(* Logix 5000 project; controller STAT 1756-L72 rev 20.12; software revision 20.04; part 29 of 34 *)
(* tags used below, declared in another part *)
   B3 : DINT[35];
   N20 : DINT[50];
   N7 : DINT[150];
   N9 : DINT[200];
   T4 : TIMER[100];
   comm : BOOL;
   L1_stat : DINT[20];
   L2_STAT : DINT[20];
   L3_STAT : DINT[20];
   lancystock1 : DINT;
   lancystock2 : DINT;
   N : INT[255];
   stat_L1 : DINT[20];
   STAT_L2 : DINT[20];
   STAT_L3 : DINT[20];
(* LANCY, continued *)

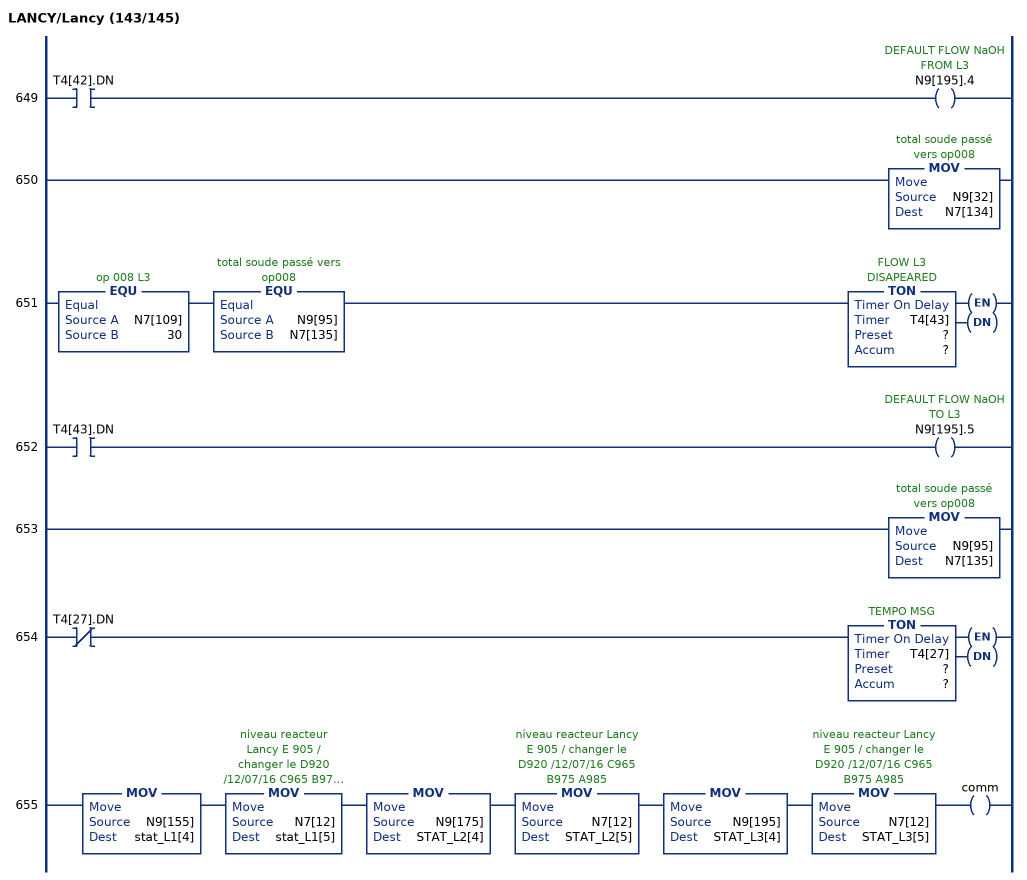
   649: XIC(T4[42].DN)OTE(N9[195].4);
   650: MOV(N9[32],N7[134]);
   651: EQU(N7[109],30)EQU(N9[95],N7[135])TON(T4[43],?,?);
   652: XIC(T4[43].DN)OTE(N9[195].5);
   653: MOV(N9[95],N7[135]);
   654: XIO(T4[27].DN)TON(T4[27],?,?);
   655: MOV(N9[155],stat_L1[4])MOV(N7[12],stat_L1[5])MOV(N9[175],STAT_L2[4])MOV(N7[12],STAT_L2[5])MOV(N9[195],STAT_L3[4])MOV(N7[12],STAT_L3[5])OTE(comm);
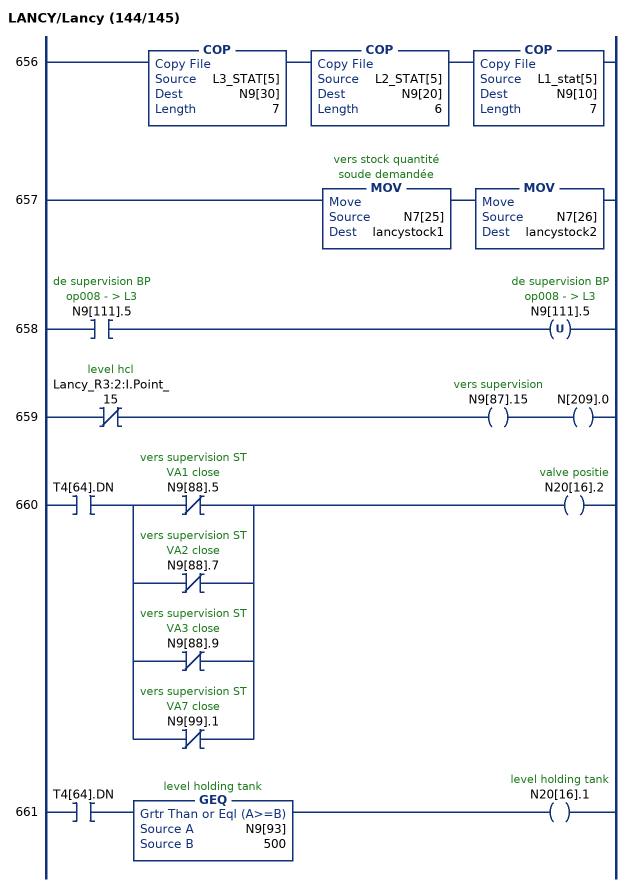
   656: COP(L3_STAT[5],N9[30],7)COP(L2_STAT[5],N9[20],6)COP(L1_stat[5],N9[10],7);
   657: MOV(N7[25],lancystock1)MOV(N7[26],lancystock2);
   658: XIC(N9[111].5)OTU(N9[111].5);
   659: XIO(Lancy_R3:2:I.Point_15)OTE(N9[87].15)OTE(N[209].0);
   660: XIC(T4[64].DN)[XIO(N9[88].5) ,XIO(N9[88].7) ,XIO(N9[88].9) ,XIO(N9[99].1) ]OTE(N20[16].2);
   661: XIC(T4[64].DN)GEQ(N9[93],500)OTE(N20[16].1);
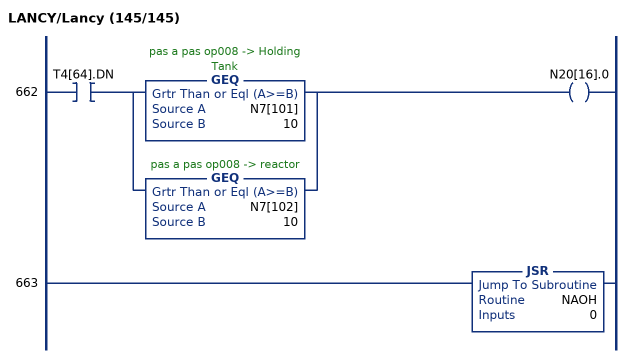
   662: XIC(T4[64].DN)[GEQ(N7[101],10) ,GEQ(N7[102],10) ]OTE(N20[16].0);
   663: JSR(NAOH,0);
END_ROUTINE

ROUTINE lancy_ALARMING   (* ladder *)
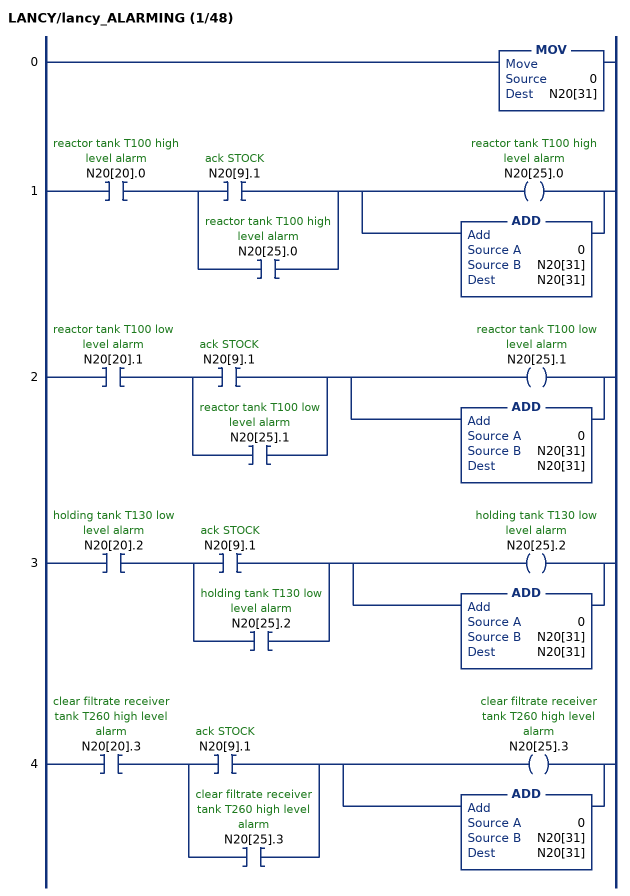
   0: MOV(0,N20[31]);
   1: XIC(N20[20].0)[XIC(N20[9].1) ,XIC(N20[25].0) ][OTE(N20[25].0) ,ADD(0,N20[31],N20[31]) ];
   2: XIC(N20[20].1)[XIC(N20[9].1) ,XIC(N20[25].1) ][OTE(N20[25].1) ,ADD(0,N20[31],N20[31]) ];
   3: XIC(N20[20].2)[XIC(N20[9].1) ,XIC(N20[25].2) ][OTE(N20[25].2) ,ADD(0,N20[31],N20[31]) ];
   4: XIC(N20[20].3)[XIC(N20[9].1) ,XIC(N20[25].3) ][OTE(N20[25].3) ,ADD(0,N20[31],N20[31]) ];
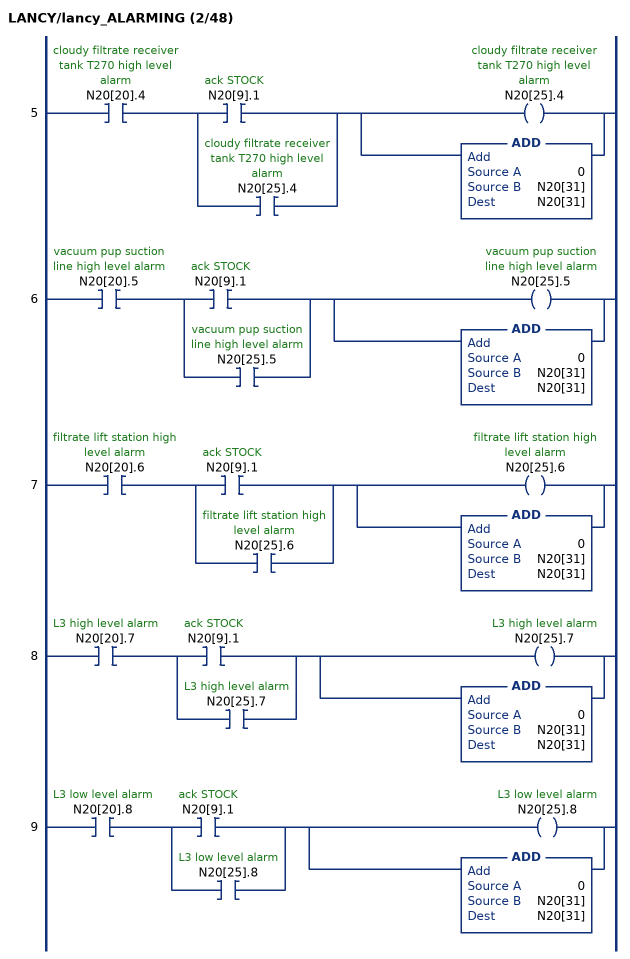
   5: XIC(N20[20].4)[XIC(N20[9].1) ,XIC(N20[25].4) ][OTE(N20[25].4) ,ADD(0,N20[31],N20[31]) ];
   6: XIC(N20[20].5)[XIC(N20[9].1) ,XIC(N20[25].5) ][OTE(N20[25].5) ,ADD(0,N20[31],N20[31]) ];
   7: XIC(N20[20].6)[XIC(N20[9].1) ,XIC(N20[25].6) ][OTE(N20[25].6) ,ADD(0,N20[31],N20[31]) ];
   8: XIC(N20[20].7)[XIC(N20[9].1) ,XIC(N20[25].7) ][OTE(N20[25].7) ,ADD(0,N20[31],N20[31]) ];
   9: XIC(N20[20].8)[XIC(N20[9].1) ,XIC(N20[25].8) ][OTE(N20[25].8) ,ADD(0,N20[31],N20[31]) ];
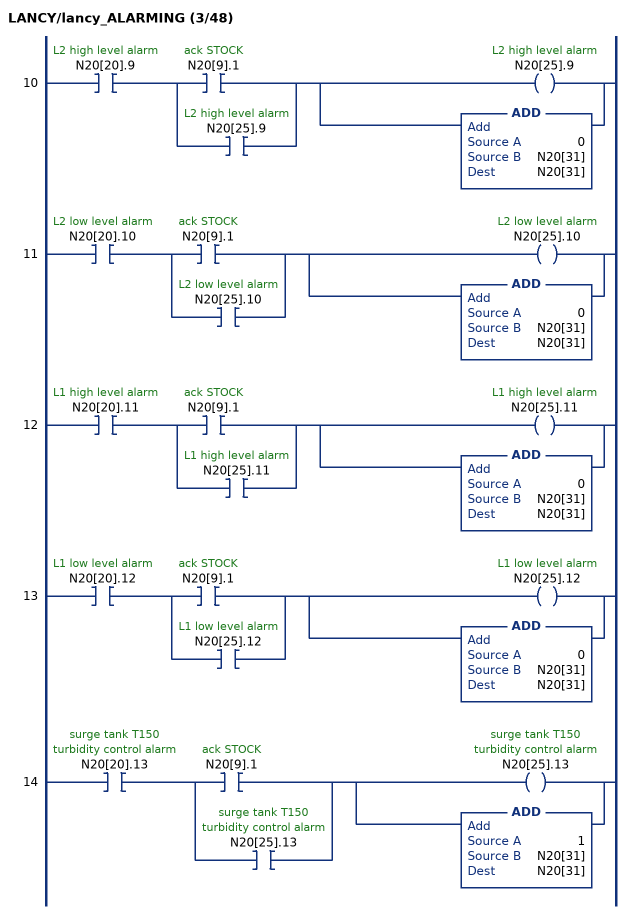
   10: XIC(N20[20].9)[XIC(N20[9].1) ,XIC(N20[25].9) ][OTE(N20[25].9) ,ADD(0,N20[31],N20[31]) ];
   11: XIC(N20[20].10)[XIC(N20[9].1) ,XIC(N20[25].10) ][OTE(N20[25].10) ,ADD(0,N20[31],N20[31]) ];
   12: XIC(N20[20].11)[XIC(N20[9].1) ,XIC(N20[25].11) ][OTE(N20[25].11) ,ADD(0,N20[31],N20[31]) ];
   13: XIC(N20[20].12)[XIC(N20[9].1) ,XIC(N20[25].12) ][OTE(N20[25].12) ,ADD(0,N20[31],N20[31]) ];
   14: XIC(N20[20].13)[XIC(N20[9].1) ,XIC(N20[25].13) ][OTE(N20[25].13) ,ADD(1,N20[31],N20[31]) ];
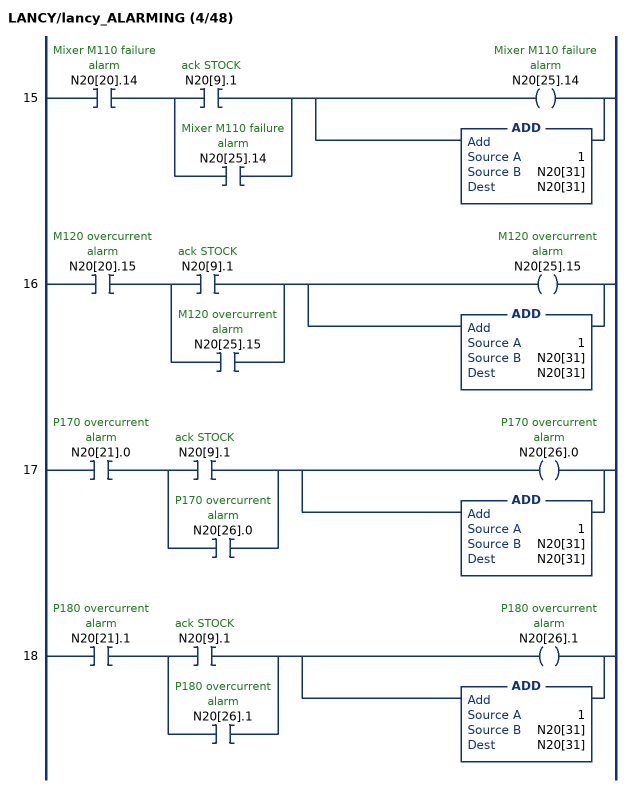
   15: XIC(N20[20].14)[XIC(N20[9].1) ,XIC(N20[25].14) ][OTE(N20[25].14) ,ADD(1,N20[31],N20[31]) ];
   16: XIC(N20[20].15)[XIC(N20[9].1) ,XIC(N20[25].15) ][OTE(N20[25].15) ,ADD(1,N20[31],N20[31]) ];
   17: XIC(N20[21].0)[XIC(N20[9].1) ,XIC(N20[26].0) ][OTE(N20[26].0) ,ADD(1,N20[31],N20[31]) ];
   18: XIC(N20[21].1)[XIC(N20[9].1) ,XIC(N20[26].1) ][OTE(N20[26].1) ,ADD(1,N20[31],N20[31]) ];
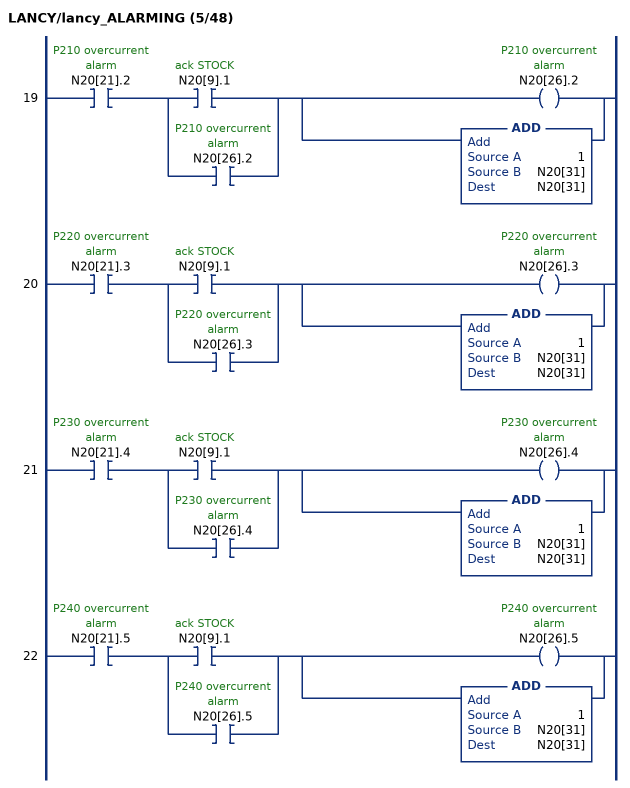
   19: XIC(N20[21].2)[XIC(N20[9].1) ,XIC(N20[26].2) ][OTE(N20[26].2) ,ADD(1,N20[31],N20[31]) ];
   20: XIC(N20[21].3)[XIC(N20[9].1) ,XIC(N20[26].3) ][OTE(N20[26].3) ,ADD(1,N20[31],N20[31]) ];
   21: XIC(N20[21].4)[XIC(N20[9].1) ,XIC(N20[26].4) ][OTE(N20[26].4) ,ADD(1,N20[31],N20[31]) ];
   22: XIC(N20[21].5)[XIC(N20[9].1) ,XIC(N20[26].5) ][OTE(N20[26].5) ,ADD(1,N20[31],N20[31]) ];
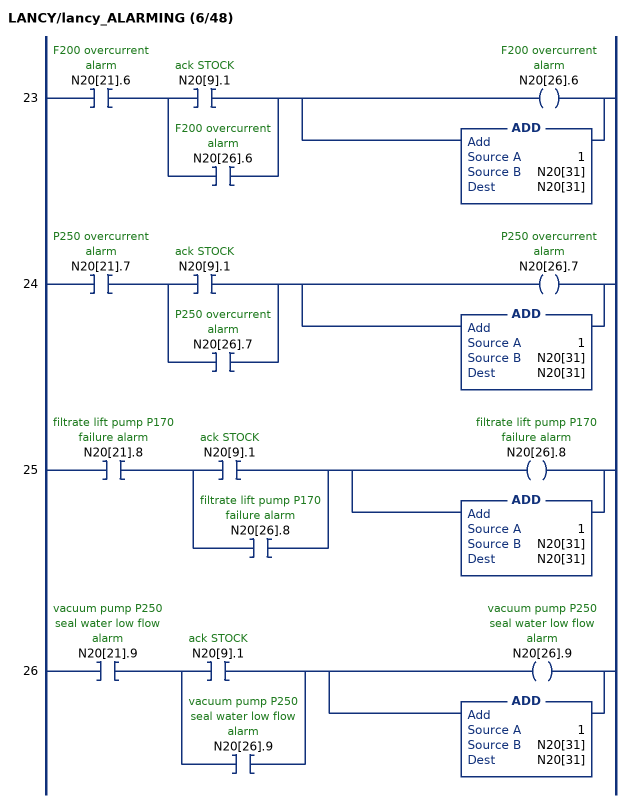
   23: XIC(N20[21].6)[XIC(N20[9].1) ,XIC(N20[26].6) ][OTE(N20[26].6) ,ADD(1,N20[31],N20[31]) ];
   24: XIC(N20[21].7)[XIC(N20[9].1) ,XIC(N20[26].7) ][OTE(N20[26].7) ,ADD(1,N20[31],N20[31]) ];
   25: XIC(N20[21].8)[XIC(N20[9].1) ,XIC(N20[26].8) ][OTE(N20[26].8) ,ADD(1,N20[31],N20[31]) ];
   26: XIC(N20[21].9)[XIC(N20[9].1) ,XIC(N20[26].9) ][OTE(N20[26].9) ,ADD(1,N20[31],N20[31]) ];
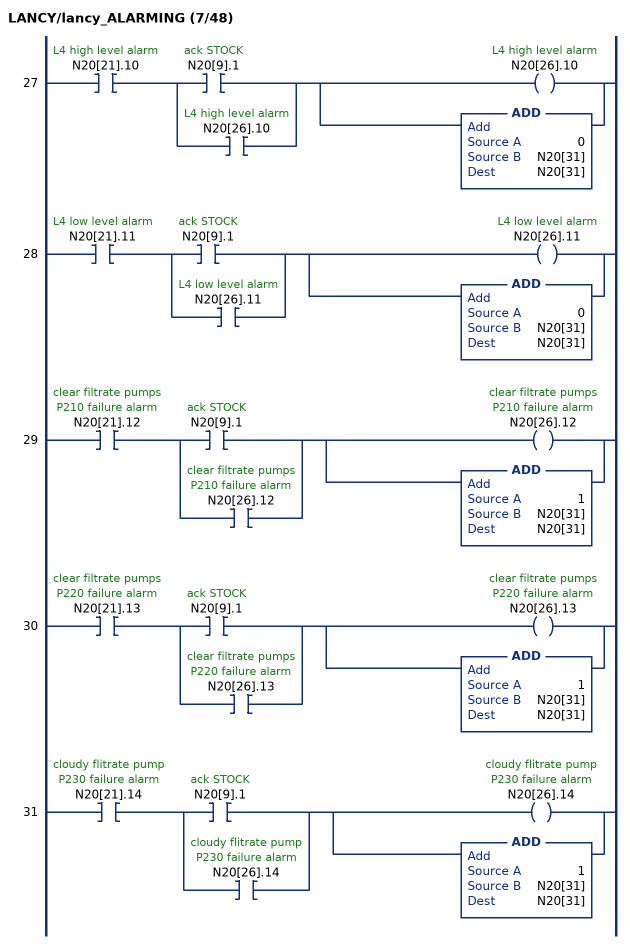
   27: XIC(N20[21].10)[XIC(N20[9].1) ,XIC(N20[26].10) ][OTE(N20[26].10) ,ADD(0,N20[31],N20[31]) ];
   28: XIC(N20[21].11)[XIC(N20[9].1) ,XIC(N20[26].11) ][OTE(N20[26].11) ,ADD(0,N20[31],N20[31]) ];
   29: XIC(N20[21].12)[XIC(N20[9].1) ,XIC(N20[26].12) ][OTE(N20[26].12) ,ADD(1,N20[31],N20[31]) ];
   30: XIC(N20[21].13)[XIC(N20[9].1) ,XIC(N20[26].13) ][OTE(N20[26].13) ,ADD(1,N20[31],N20[31]) ];
   31: XIC(N20[21].14)[XIC(N20[9].1) ,XIC(N20[26].14) ][OTE(N20[26].14) ,ADD(1,N20[31],N20[31]) ];
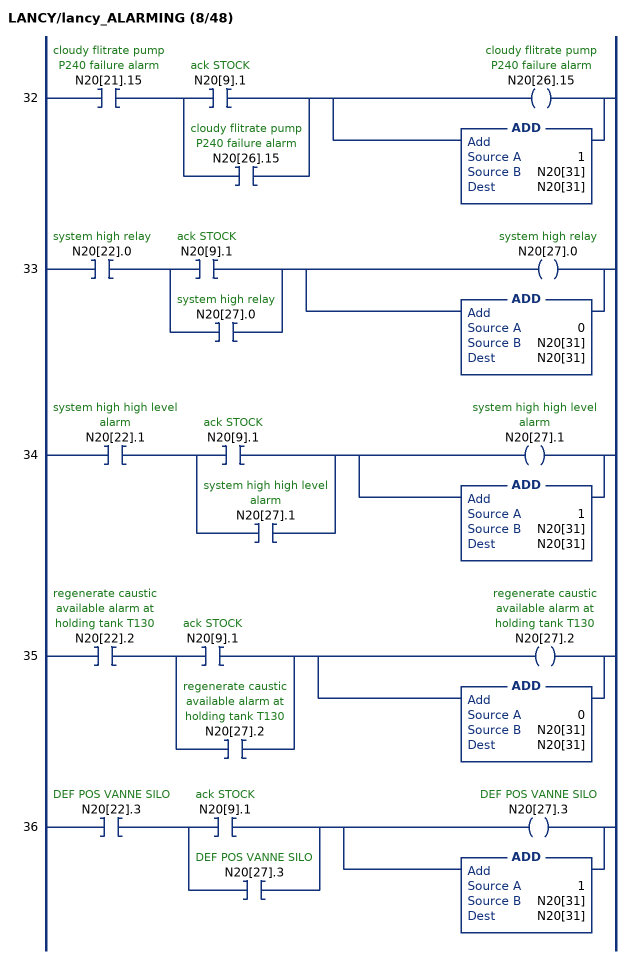
   32: XIC(N20[21].15)[XIC(N20[9].1) ,XIC(N20[26].15) ][OTE(N20[26].15) ,ADD(1,N20[31],N20[31]) ];
   33: XIC(N20[22].0)[XIC(N20[9].1) ,XIC(N20[27].0) ][OTE(N20[27].0) ,ADD(0,N20[31],N20[31]) ];
   34: XIC(N20[22].1)[XIC(N20[9].1) ,XIC(N20[27].1) ][OTE(N20[27].1) ,ADD(1,N20[31],N20[31]) ];
   35: XIC(N20[22].2)[XIC(N20[9].1) ,XIC(N20[27].2) ][OTE(N20[27].2) ,ADD(0,N20[31],N20[31]) ];
   36: XIC(N20[22].3)[XIC(N20[9].1) ,XIC(N20[27].3) ][OTE(N20[27].3) ,ADD(1,N20[31],N20[31]) ];
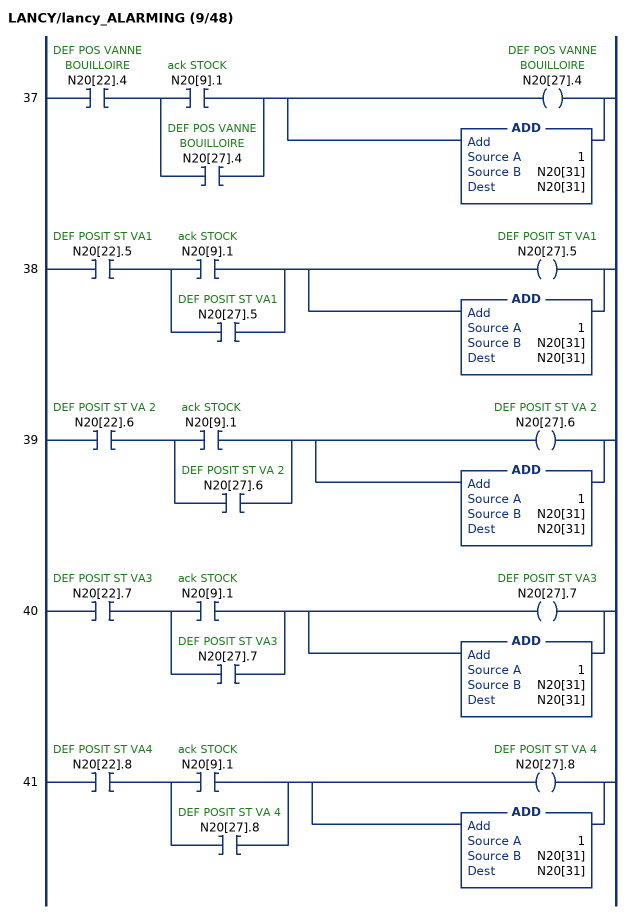
   37: XIC(N20[22].4)[XIC(N20[9].1) ,XIC(N20[27].4) ][OTE(N20[27].4) ,ADD(1,N20[31],N20[31]) ];
   38: XIC(N20[22].5)[XIC(N20[9].1) ,XIC(N20[27].5) ][OTE(N20[27].5) ,ADD(1,N20[31],N20[31]) ];
   39: XIC(N20[22].6)[XIC(N20[9].1) ,XIC(N20[27].6) ][OTE(N20[27].6) ,ADD(1,N20[31],N20[31]) ];
   40: XIC(N20[22].7)[XIC(N20[9].1) ,XIC(N20[27].7) ][OTE(N20[27].7) ,ADD(1,N20[31],N20[31]) ];
   41: XIC(N20[22].8)[XIC(N20[9].1) ,XIC(N20[27].8) ][OTE(N20[27].8) ,ADD(1,N20[31],N20[31]) ];
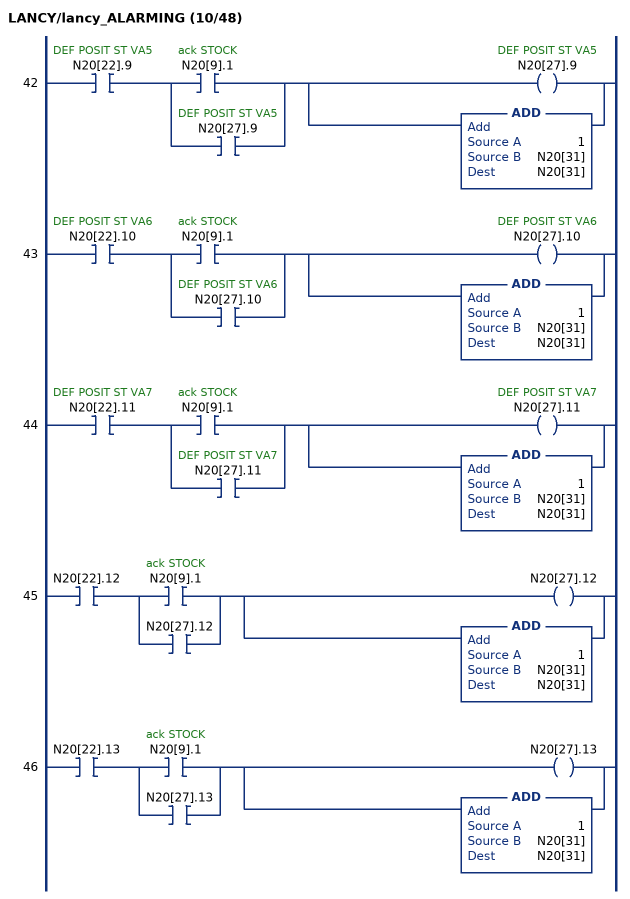
   42: XIC(N20[22].9)[XIC(N20[9].1) ,XIC(N20[27].9) ][OTE(N20[27].9) ,ADD(1,N20[31],N20[31]) ];
   43: XIC(N20[22].10)[XIC(N20[9].1) ,XIC(N20[27].10) ][OTE(N20[27].10) ,ADD(1,N20[31],N20[31]) ];
   44: XIC(N20[22].11)[XIC(N20[9].1) ,XIC(N20[27].11) ][OTE(N20[27].11) ,ADD(1,N20[31],N20[31]) ];
   45: XIC(N20[22].12)[XIC(N20[9].1) ,XIC(N20[27].12) ][OTE(N20[27].12) ,ADD(1,N20[31],N20[31]) ];
   46: XIC(N20[22].13)[XIC(N20[9].1) ,XIC(N20[27].13) ][OTE(N20[27].13) ,ADD(1,N20[31],N20[31]) ];
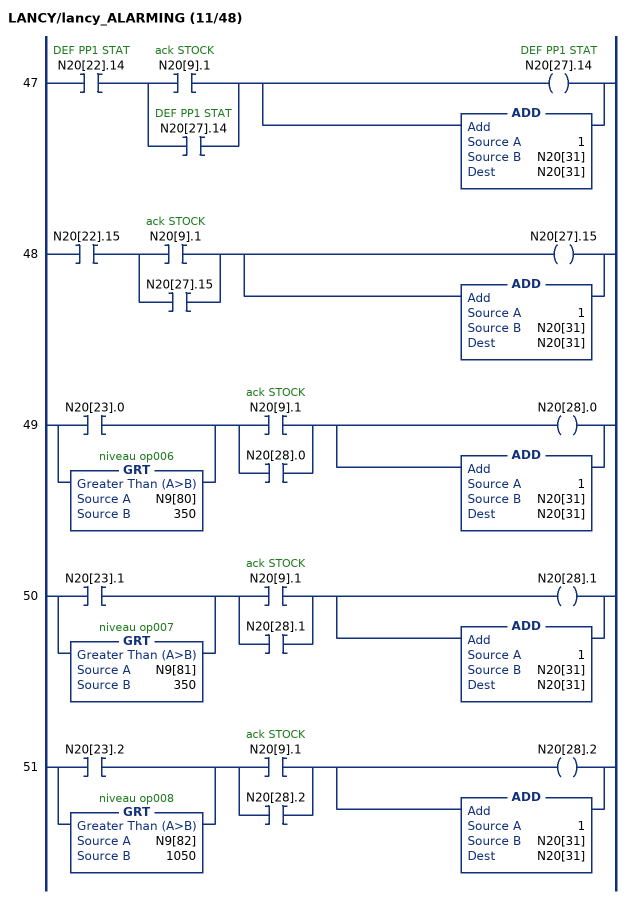
   47: XIC(N20[22].14)[XIC(N20[9].1) ,XIC(N20[27].14) ][OTE(N20[27].14) ,ADD(1,N20[31],N20[31]) ];
   48: XIC(N20[22].15)[XIC(N20[9].1) ,XIC(N20[27].15) ][OTE(N20[27].15) ,ADD(1,N20[31],N20[31]) ];
   49: [XIC(N20[23].0) ,GRT(N9[80],350) ][XIC(N20[9].1) ,XIC(N20[28].0) ][OTE(N20[28].0) ,ADD(1,N20[31],N20[31]) ];
   50: [XIC(N20[23].1) ,GRT(N9[81],350) ][XIC(N20[9].1) ,XIC(N20[28].1) ][OTE(N20[28].1) ,ADD(1,N20[31],N20[31]) ];
   51: [XIC(N20[23].2) ,GRT(N9[82],1050) ][XIC(N20[9].1) ,XIC(N20[28].2) ][OTE(N20[28].2) ,ADD(1,N20[31],N20[31]) ];
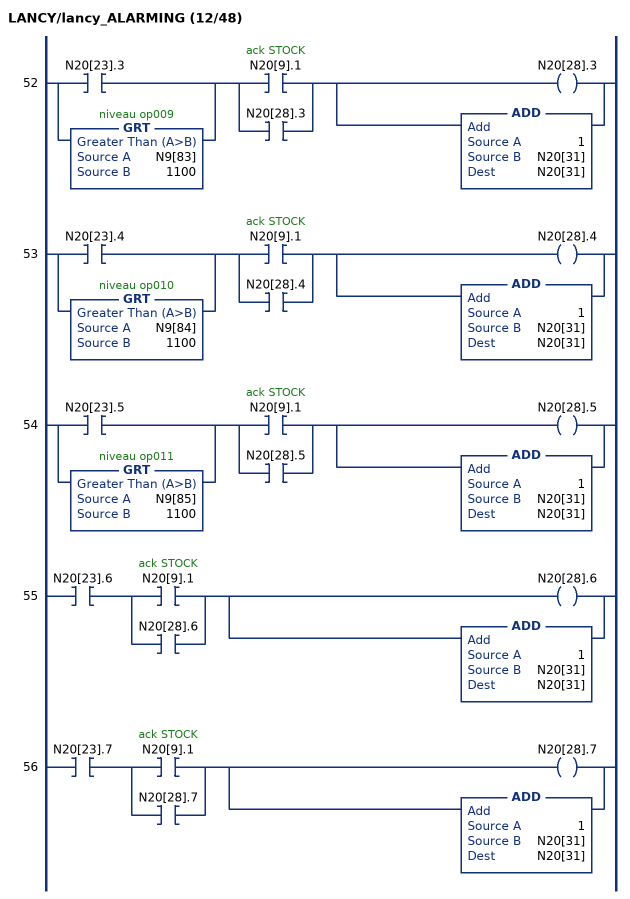
   52: [XIC(N20[23].3) ,GRT(N9[83],1100) ][XIC(N20[9].1) ,XIC(N20[28].3) ][OTE(N20[28].3) ,ADD(1,N20[31],N20[31]) ];
   53: [XIC(N20[23].4) ,GRT(N9[84],1100) ][XIC(N20[9].1) ,XIC(N20[28].4) ][OTE(N20[28].4) ,ADD(1,N20[31],N20[31]) ];
   54: [XIC(N20[23].5) ,GRT(N9[85],1100) ][XIC(N20[9].1) ,XIC(N20[28].5) ][OTE(N20[28].5) ,ADD(1,N20[31],N20[31]) ];
   55: XIC(N20[23].6)[XIC(N20[9].1) ,XIC(N20[28].6) ][OTE(N20[28].6) ,ADD(1,N20[31],N20[31]) ];
   56: XIC(N20[23].7)[XIC(N20[9].1) ,XIC(N20[28].7) ][OTE(N20[28].7) ,ADD(1,N20[31],N20[31]) ];
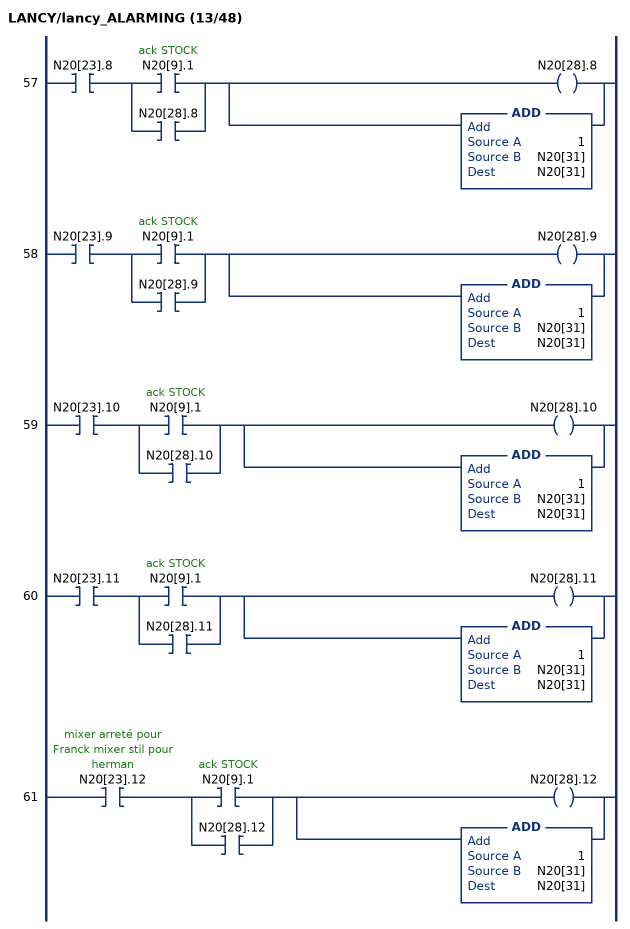
   57: XIC(N20[23].8)[XIC(N20[9].1) ,XIC(N20[28].8) ][OTE(N20[28].8) ,ADD(1,N20[31],N20[31]) ];
   58: XIC(N20[23].9)[XIC(N20[9].1) ,XIC(N20[28].9) ][OTE(N20[28].9) ,ADD(1,N20[31],N20[31]) ];
   59: XIC(N20[23].10)[XIC(N20[9].1) ,XIC(N20[28].10) ][OTE(N20[28].10) ,ADD(1,N20[31],N20[31]) ];
   60: XIC(N20[23].11)[XIC(N20[9].1) ,XIC(N20[28].11) ][OTE(N20[28].11) ,ADD(1,N20[31],N20[31]) ];
   61: XIC(N20[23].12)[XIC(N20[9].1) ,XIC(N20[28].12) ][OTE(N20[28].12) ,ADD(1,N20[31],N20[31]) ];
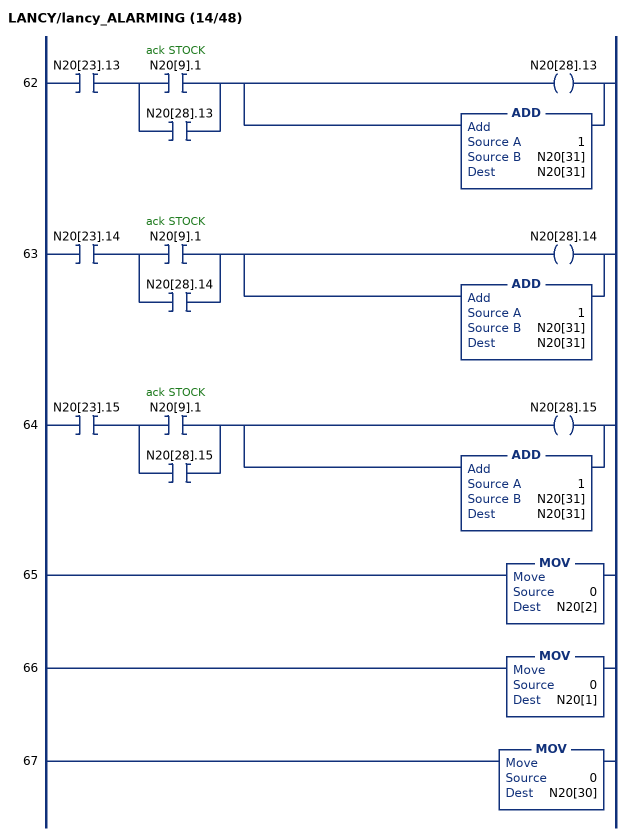
   62: XIC(N20[23].13)[XIC(N20[9].1) ,XIC(N20[28].13) ][OTE(N20[28].13) ,ADD(1,N20[31],N20[31]) ];
   63: XIC(N20[23].14)[XIC(N20[9].1) ,XIC(N20[28].14) ][OTE(N20[28].14) ,ADD(1,N20[31],N20[31]) ];
   64: XIC(N20[23].15)[XIC(N20[9].1) ,XIC(N20[28].15) ][OTE(N20[28].15) ,ADD(1,N20[31],N20[31]) ];
   65: MOV(0,N20[2]);
   66: MOV(0,N20[1]);
   67: MOV(0,N20[30]);
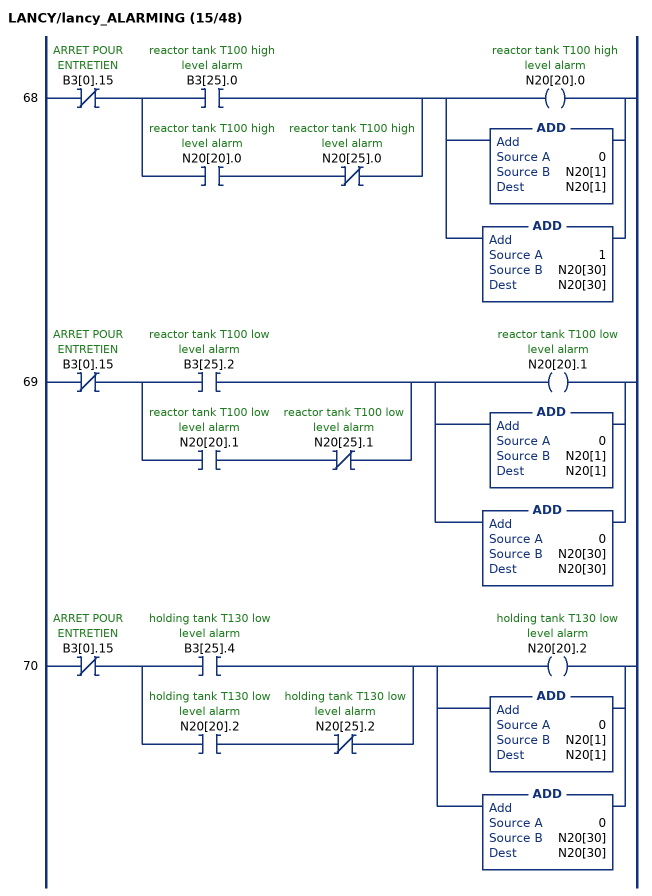
   68: XIO(B3[0].15)[XIC(B3[25].0) ,XIC(N20[20].0) XIO(N20[25].0) ][OTE(N20[20].0) ,ADD(0,N20[1],N20[1]) ,ADD(1,N20[30],N20[30]) ];
   69: XIO(B3[0].15)[XIC(B3[25].2) ,XIC(N20[20].1) XIO(N20[25].1) ][OTE(N20[20].1) ,ADD(0,N20[1],N20[1]) ,ADD(0,N20[30],N20[30]) ];
   70: XIO(B3[0].15)[XIC(B3[25].4) ,XIC(N20[20].2) XIO(N20[25].2) ][OTE(N20[20].2) ,ADD(0,N20[1],N20[1]) ,ADD(0,N20[30],N20[30]) ];
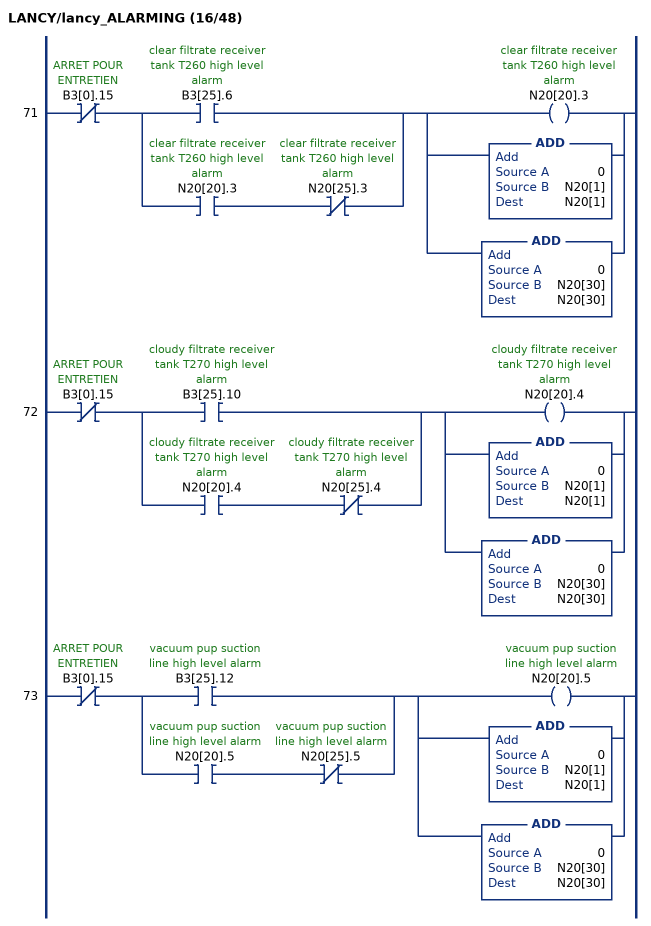
   71: XIO(B3[0].15)[XIC(B3[25].6) ,XIC(N20[20].3) XIO(N20[25].3) ][OTE(N20[20].3) ,ADD(0,N20[1],N20[1]) ,ADD(0,N20[30],N20[30]) ];
   72: XIO(B3[0].15)[XIC(B3[25].10) ,XIC(N20[20].4) XIO(N20[25].4) ][OTE(N20[20].4) ,ADD(0,N20[1],N20[1]) ,ADD(0,N20[30],N20[30]) ];
   73: XIO(B3[0].15)[XIC(B3[25].12) ,XIC(N20[20].5) XIO(N20[25].5) ][OTE(N20[20].5) ,ADD(0,N20[1],N20[1]) ,ADD(0,N20[30],N20[30]) ];
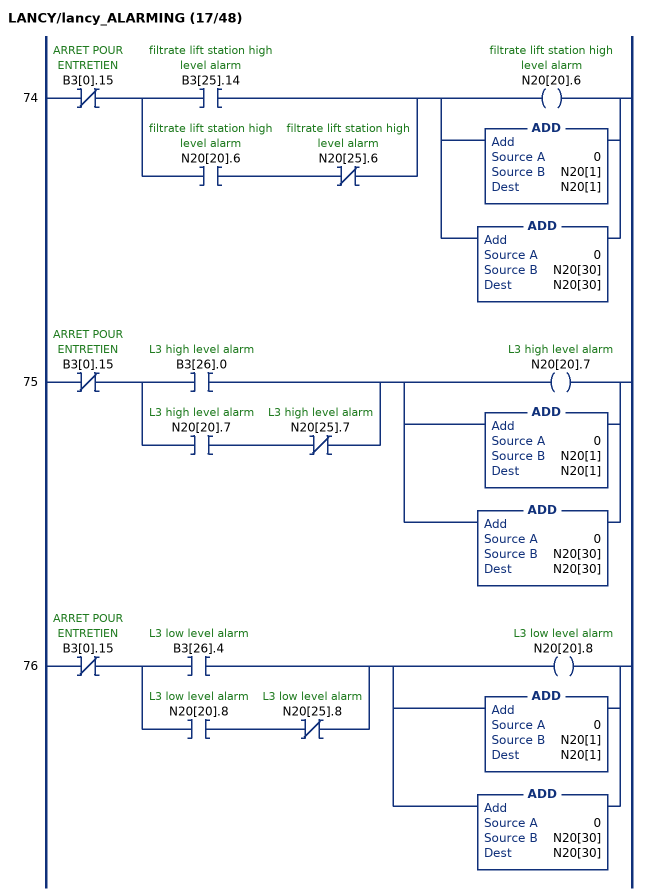
   74: XIO(B3[0].15)[XIC(B3[25].14) ,XIC(N20[20].6) XIO(N20[25].6) ][OTE(N20[20].6) ,ADD(0,N20[1],N20[1]) ,ADD(0,N20[30],N20[30]) ];
   75: XIO(B3[0].15)[XIC(B3[26].0) ,XIC(N20[20].7) XIO(N20[25].7) ][OTE(N20[20].7) ,ADD(0,N20[1],N20[1]) ,ADD(0,N20[30],N20[30]) ];
   76: XIO(B3[0].15)[XIC(B3[26].4) ,XIC(N20[20].8) XIO(N20[25].8) ][OTE(N20[20].8) ,ADD(0,N20[1],N20[1]) ,ADD(0,N20[30],N20[30]) ];
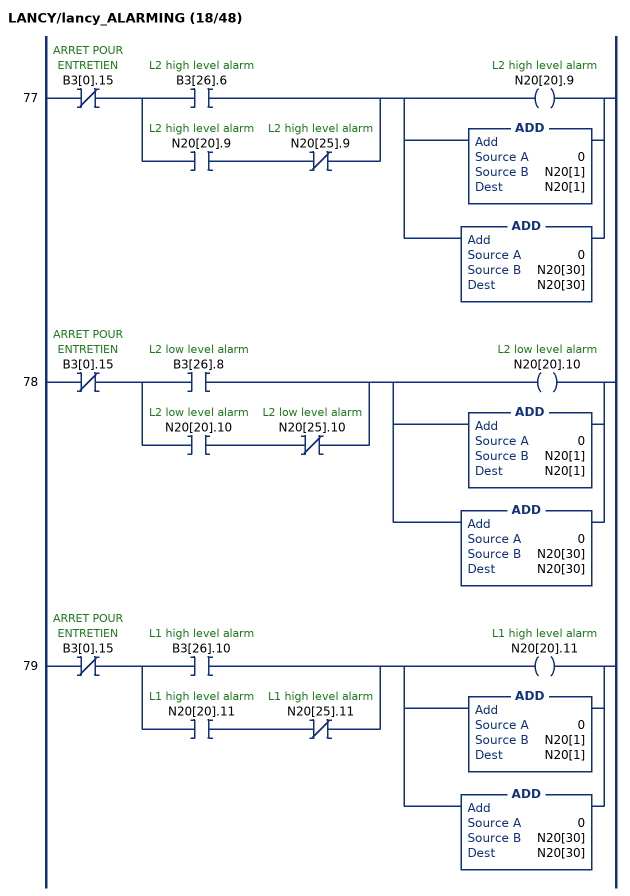
   77: XIO(B3[0].15)[XIC(B3[26].6) ,XIC(N20[20].9) XIO(N20[25].9) ][OTE(N20[20].9) ,ADD(0,N20[1],N20[1]) ,ADD(0,N20[30],N20[30]) ];
   78: XIO(B3[0].15)[XIC(B3[26].8) ,XIC(N20[20].10) XIO(N20[25].10) ][OTE(N20[20].10) ,ADD(0,N20[1],N20[1]) ,ADD(0,N20[30],N20[30]) ];
   79: XIO(B3[0].15)[XIC(B3[26].10) ,XIC(N20[20].11) XIO(N20[25].11) ][OTE(N20[20].11) ,ADD(0,N20[1],N20[1]) ,ADD(0,N20[30],N20[30]) ];
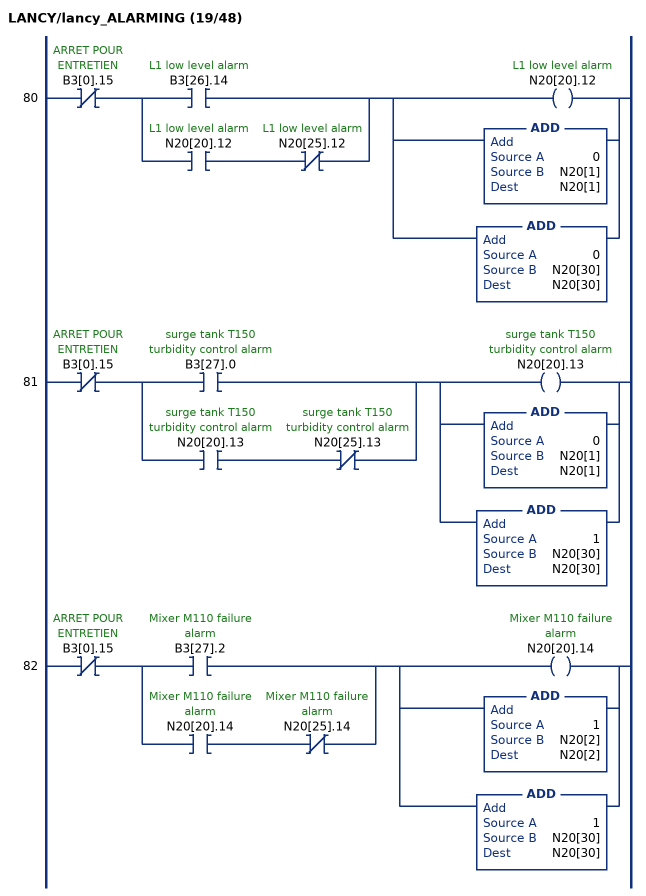
   80: XIO(B3[0].15)[XIC(B3[26].14) ,XIC(N20[20].12) XIO(N20[25].12) ][OTE(N20[20].12) ,ADD(0,N20[1],N20[1]) ,ADD(0,N20[30],N20[30]) ];
   81: XIO(B3[0].15)[XIC(B3[27].0) ,XIC(N20[20].13) XIO(N20[25].13) ][OTE(N20[20].13) ,ADD(0,N20[1],N20[1]) ,ADD(1,N20[30],N20[30]) ];
   82: XIO(B3[0].15)[XIC(B3[27].2) ,XIC(N20[20].14) XIO(N20[25].14) ][OTE(N20[20].14) ,ADD(1,N20[2],N20[2]) ,ADD(1,N20[30],N20[30]) ];
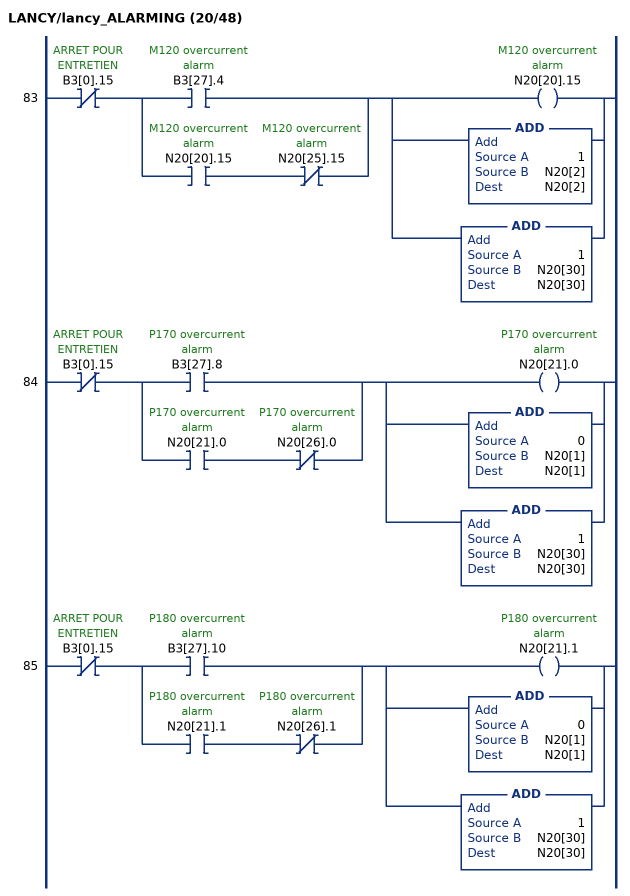
   83: XIO(B3[0].15)[XIC(B3[27].4) ,XIC(N20[20].15) XIO(N20[25].15) ][OTE(N20[20].15) ,ADD(1,N20[2],N20[2]) ,ADD(1,N20[30],N20[30]) ];
   84: XIO(B3[0].15)[XIC(B3[27].8) ,XIC(N20[21].0) XIO(N20[26].0) ][OTE(N20[21].0) ,ADD(0,N20[1],N20[1]) ,ADD(1,N20[30],N20[30]) ];
   85: XIO(B3[0].15)[XIC(B3[27].10) ,XIC(N20[21].1) XIO(N20[26].1) ][OTE(N20[21].1) ,ADD(0,N20[1],N20[1]) ,ADD(1,N20[30],N20[30]) ];
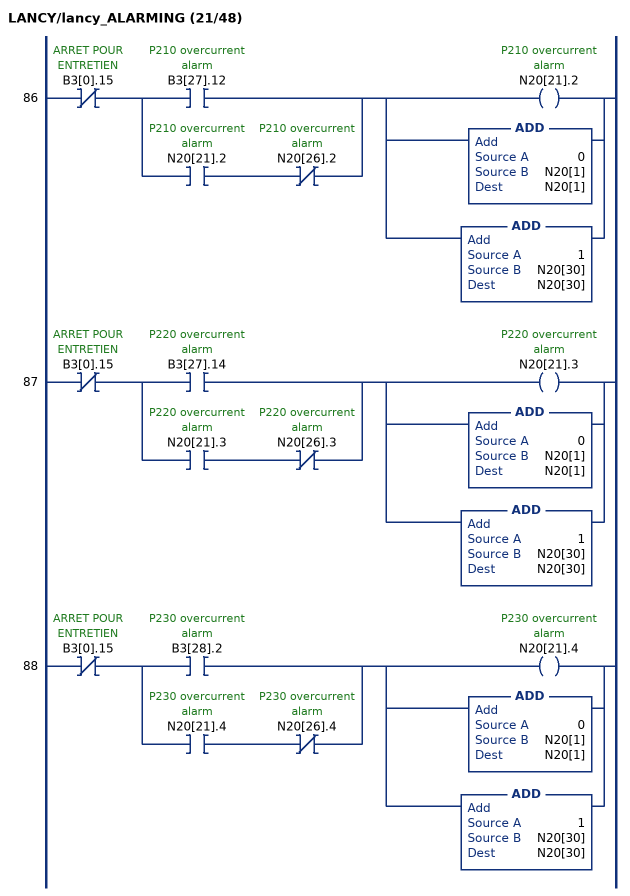
   86: XIO(B3[0].15)[XIC(B3[27].12) ,XIC(N20[21].2) XIO(N20[26].2) ][OTE(N20[21].2) ,ADD(0,N20[1],N20[1]) ,ADD(1,N20[30],N20[30]) ];
   87: XIO(B3[0].15)[XIC(B3[27].14) ,XIC(N20[21].3) XIO(N20[26].3) ][OTE(N20[21].3) ,ADD(0,N20[1],N20[1]) ,ADD(1,N20[30],N20[30]) ];
   88: XIO(B3[0].15)[XIC(B3[28].2) ,XIC(N20[21].4) XIO(N20[26].4) ][OTE(N20[21].4) ,ADD(0,N20[1],N20[1]) ,ADD(1,N20[30],N20[30]) ];
